// TwinCAT 3 PLC project
// libraries:
//   Tc2_Standard, * (Beckhoff Automation GmbH)
//   Tc2_System, * (Beckhoff Automation GmbH)
//   Tc3_Module, * (Beckhoff Automation GmbH)
//   TcUnit, * (www.tcunit.org)
// project tree:
//   TESTS/ PRG_TESTS.TcPOU
//   TESTS/Test suites/ FB_SUT_Tests.TcPOU

// ---- TESTS/PRG_TESTS.TcPOU
PROGRAM PRG_TESTS

(* Instantiate test suites here. Naming convention for tests should be a suffix with _Tests.
Good practice for creating test methods is to end them with _test as well. *)
VAR
	fbSUT_Tests	: FB_SUT_Tests;
END_VAR

// Run tests in parallel
//TcUnit.RUN();

// Run tests in sequence, one after the other.
TcUnit.RUN_IN_SEQUENCE();

END_PROGRAM

// ---- TESTS/Test suites/FB_SUT_Tests.TcPOU
// Subject under test
FUNCTION_BLOCK FB_SUT_Tests EXTENDS FB_TestSuite

// Create instance variables that will be accesible for all tests
VAR
END_VAR

// Call your test methods here
TestXX_Template();

METHOD PRIVATE TestXX_Template

(* Instanced variables are VERY useful for writing tests since tests are run in paralel (by default).
By instantiating local variables that are not placed on the same stack as method (values are retained between calls)
you make sure that the SUT is not changed by some other test. *)
VAR_INST
	
END_VAR

// Place temporary variables here
VAR
	
END_VAR
// The name of the test, is the same as method name!
// Use this for paralel unit tests
// TcUnit.TEST('TestXX_Template');

// Use this for running tests in sequence
IF TcUnit.TEST_ORDERED('TestXX_Template') THEN
	// Do your assertions here...
	AssertTrue(
		Condition := FALSE, 
		Message := 'Implement tests!');

	TcUnit.TEST_FINISHED();
END_IF
END_METHOD

END_FUNCTION_BLOCK
